{attribute 'pack_mode' := '1'}
TYPE TRunDataTable :
STRUCT
	aTPartData						: ARRAY[0..1,0..1,0..1] OF TPartData;	(*Layering, Layering Offset, Side *)
	iGiveTakeLayeringPosition			: INT;
	iGiveTakeLayeringOffsetPosition	: INT;
	eTableSide						: TTableSide;
END_STRUCT
END_TYPE

(* stored: Version 1.1.0.1, ProductVersion 3.1.4022.12
   DUT TRunDataTable: Id {52c84f48-ca66-47bc-8da7-62eaaa0f52d0} *)
